// TIA Portal V20 export
TYPE "typeSequenceControlNode_topTapeLoading"
// stored: Namespace Unit1.Em3
   STRUCT
      jobs : "LAF_typeJobs";
      sequence : "LAF_typeSequence";
      selectJobStatus { S7_SetPoint := 'True'} : Array[0..10] of "LAF_typeJobStatus";
      "step" : "LER_typeStep";
      jobInterface : "Unit1.Em3.typeSequenceControlNodeJobInterface_topTapeLoading";
      homeCheck : "Unit1.Em3.typeSequenceControlNodeHomeCheck_topTapeLoading";
   END_STRUCT;
   // // "step".action1[101] : Step[101] : JOB[1] Condition
   // // "step".action1[110] : Step[110] : Top Tape Loading Backward
   // // "step".action1[120] : Step[120] : Top Tape Loading Clamp Open
   // // "step".action1[130] : Step[130] : Top Tape Cutter Up
   // // "step".action1[140] : Step[140] : Top Tape Cutter Clamp Down
   // // "step".action1[150] : Step[150] : Top Tape Tension Backward
   // // "step".action1[190] : Step[190] : JOB[1] Step End
   // // "step".action1[201] : Step[201] : JOB[2] Condition
   // // "step".action1[210] : Step[210] : Top Tape Loading Forward & Tension Backward
   // // "step".action1[220] : Step[220] : Top Tape Clamp Close
   // // "step".action1[230] : Step[230] : Top Tape Cutter Clamp Up
   // // "step".action1[240] : Step[240] : Top Tape Loading Backward & Tension Forward
   // // "step".action1[250] : Step[250] : Top Tape Cutter Clamp Down
   // // "step".action1[260] : Step[260] : Top Tape Tension Backward
   // // "step".action1[290] : Step[290] : JOB[2] Step End
   // // "step".transition1[101] : Step[101] : JOB[1] Condition
   // // "step".transition1[110] : Step[110] : Top Tape Loading Backward
   // // "step".transition1[120] : Step[120] : Top Tape Loading Clamp Open
   // // "step".transition1[130] : Step[130] : Top Tape Cutter Up
   // // "step".transition1[140] : Step[140] : Top Tape Cutter Clamp Down
   // // "step".transition1[150] : Step[150] : Top Tape Tension Backward
   // // "step".transition1[190] : Step[190] : JOB[1] Step End
   // // "step".transition1[201] : Step[201] : JOB[2] Condition
   // // "step".transition1[210] : Step[210] : Top Tape Loading Forward & Tension Backward
   // // "step".transition1[220] : Step[220] : Top Tape Clamp Close
   // // "step".transition1[230] : Step[230] : Top Tape Cutter Clamp Up
   // // "step".transition1[240] : Step[240] : Top Tape Loading Backward & Tension Forward
   // // "step".transition1[250] : Step[250] : Top Tape Cutter Clamp Down
   // // "step".transition1[260] : Step[260] : Top Tape Tension Backward
   // // "step".transition1[290] : Step[290] : JOB[2] Step End
END_TYPE
